TYPE HMIRFIDDataInterface :
STRUCT
	SingleReadValue	:	WORD;
	SingleWriteValue	:	WORD;
	AllReadData	:	ARRAY[0..127] OF WORD;
	AllWriteData	:	ARRAY[0..127] OF WORD;
END_STRUCT
END_TYPE

(* stored: Version 1.1.0.1
   DUT HMIRFIDDataInterface: Id {273f5c2b-c243-47cc-a622-124862ad9d1e} *)
